(* IEC 61131-3 sources: axftcmlib/src/Sortingline, 10 files *)

(* ---- ISortingline.st ---- *)
NAMESPACE Simatic.Ax.axftcmlib
    INTERFACE ISortingline
        METHOD SlMoveToColorsensor
        END_METHOD
        METHOD SlDetectColor : Bool
        END_METHOD
        METHOD SlMoveToSensor
        END_METHOD
        METHOD SlClearConveyor
        END_METHOD

    END_INTERFACE
END_NAMESPACE

(* ---- Sl1StateIdle.st ---- *)
USING Simatic.Ax.StateFramework;
//SOrtingline is ready for the next Element to be sorted
NAMESPACE Simatic.Ax.axftcmlib

    CLASS INTERNAL SlStateIdle EXTENDS State1Transition
        VAR PUBLIC //Reset
           UsedSortingline : Sortingline;
        END_VAR
        METHOD PUBLIC OVERRIDE  OnEntry
          ;
        END_METHOD
    END_CLASS

END_NAMESPACE

(* ---- Sl2StateMoveToColorSensor.st ---- *)
USING Simatic.Ax.StateFramework;
//If an element is placed infront of the first sensor, the Axis moves to the colorsensor
NAMESPACE Simatic.Ax.axftcmlib

    CLASS INTERNAL SlStateMoveToColorSensor EXTENDS State1Transition
        VAR PUBLIC
          Sortingline : ISortingline;
        END_VAR
        METHOD PUBLIC OVERRIDE  OnEntry
            Sortingline.SlMoveToColorsensor();
        END_METHOD
    END_CLASS

END_NAMESPACE

(* ---- Sl3StateDetectColor-Edit.st ---- *)
USING Simatic.Ax.StateFramework;
//if the axis is done, the sensor detects the color and puts it oput
    //->Color valid PArt will be sorted by pusher -> Path 1
    //->color invalid (=#Unknown) ->Path 2
NAMESPACE Simatic.Ax.axftcmlib

    CLASS INTERNAL SlStateDetectColor EXTENDS State2Transition
    VAR
        UsedSortingline : ISortingline;
    END_VAR
        METHOD PUBLIC OVERRIDE OnEntry
            UsedSortingline.SlDetectColor();
        END_METHOD
    END_CLASS

END_NAMESPACE

(* ---- Sl4_1StateColorDetected.st ---- *)
USING Simatic.Ax.StateFramework;
//Valid element is transported to the next sensor
NAMESPACE Simatic.Ax.axftcmlib

    CLASS INTERNAL SlColorDetected EXTENDS State1Transition
        VAR PUBLIC //Reset
          UsedSortingline : ISortingline;
        END_VAR
        METHOD PUBLIC OVERRIDE  OnEntry
            UsedSortingline.SlMoveToSensor();
        END_METHOD
    END_CLASS

END_NAMESPACE

(* ---- Sl4_2StateColorNotDetected.st ---- *)
USING Simatic.Ax.StateFramework;

//element is thrown out of the Sortingline by the conveyor
NAMESPACE Simatic.Ax.axftcmlib

    CLASS INTERNAL SlColorNotDetected EXTENDS State1Transition
        VAR PUBLIC //Reset
          UsedSortingline : ISortingline;
        END_VAR
        METHOD PUBLIC OVERRIDE  OnEntry
            USedSOrtingline.SlClearConveyor();
        END_METHOD
    END_CLASS

END_NAMESPACE

// SlAxis : AXIS;
// SlVelocity : LREAL;
// Activetime : PULSE := (duration := LT#5.0s);//TODO Duration
// METHOD PUBLIC OVERRIDE  OnEntry
//     VAR
//         dir : INT := 0;
//         Trigger : BOOL;
//     END_VAR
//  Trigger := TRUE;
//  IF ActiveTime.output THEN
//  SlAxis.MoveVelocity(SlVelocity,dir);
//  ELSE
// SlAxis.HALT();
//  END_IF;
// END_METHOD

(* ---- Sl5_1StateChoseCylinder.st ---- *)
USING Simatic.Ax.StateFramework;

NAMESPACE Simatic.Ax.axftcmlib

    CLASS INTERNAL SlChoseCylinder EXTENDS State1Transition
        VAR PUBLIC //Reset
           SlAxis : AXIS;
           SlVelocity : LREAL;
           Sensor : BOOL;
           Color : INT;
           PosWHITE : LINT;
           PosRED : LINT;
           PosBLUE : LINT;

        END_VAR
        METHOD PUBLIC OVERRIDE  OnEntry

            VAR
                value : LINT := 0;
            END_VAR

            IF Sensor = TRUE THEN
                SlAxis.Halt();
                SlAxis.Homing(value);
                IF Color = Colors#WHITE THEN
                    SlAxis.MoveRelative(SlVelocity,PosWHITE);
                ELSIF Color = Colors#RED THEN
                    SlAxis.MoveRelative(SlVelocity, PosRED);
                ELSE
                    SlAxis.MoveRelative(SlVelocity, PosBLUE);
                END_IF;
            END_IF;

        END_METHOD
    END_CLASS

END_NAMESPACE

(* ---- Sl6_1StatePusher.st ---- *)
USING Simatic.Ax.StateFramework;

NAMESPACE Simatic.Ax.axftcmlib

    CLASS INTERNAL SlActivateCylinder EXTENDS State1Transition
        VAR PUBLIC //Reset
            CylinderWhite : PneumaticCylinder;
            CylinderRed : PneumaticCylinder;
            CylinderBlue :  PneumaticCylinder;
           Color : INT;
        END_VAR
        METHOD PUBLIC OVERRIDE  OnEntry
                IF Color = Colors#WHITE THEN
                    CylinderWhite.start();
                ELSIF Color = Colors#RED THEN
                    CylinderRed.start();
                ELSE
                    CylinderBlue.start();
                END_IF;
        END_METHOD
    END_CLASS

END_NAMESPACE

(* ---- Sl71-2SortingDone.st ---- *)
USING Simatic.Ax.StateFramework;

NAMESPACE Simatic.Ax.axftcmlib

    CLASS INTERNAL SlSortingDone EXTENDS State1Transition
        VAR PUBLIC //Reset
           SlAxis : AXIS;
        END_VAR
        METHOD PUBLIC OVERRIDE  OnEntry
               SlAxis.Halt();
        END_METHOD
    END_CLASS

END_NAMESPACE

(* ---- Sortingline.st ---- *)
USING Simatic.Ax.IO;
USING Simatic.Ax.axftcmlib;
USING Simatic.Ax.IO.Output;
USING Simatic.Ax.StateFramework;
USING System.Timer;
NAMESPACE Simatic.Ax.axftcmlib
    CLASS Sortingline EXTENDS ControlModuleAbstract IMPLEMENTS ISortingline

        VAR PUBLIC

            SlAxis : Axis;
            SlTimeProvider : TimeProvider;
            SlAxisVelocity : LREAL;
            SlAxisPositionColorSensor : LINT;
            SlAxisPositionWhite : LINT;
            SlAxisPositionRed : LINT;
            SlAxisPositionBlue : LINT;
            Homingposition : LINT := 0;
            SlColorSensor : ColorSensor;
            SlColorvalue : INT;
            ResultColor : INT;
            ColorArray : ARRAY[0..3] OF ColorRange;
            SlCompressor : PneumaticCompressor;
            SlCoilPushingWhite : IBinOutput;
            SlCoilpushingRed : IBinOutput;
            SlCoilPushingBlue : IBinOutput;
            SlSensorActivation : BOOL;
            SlSensorSorting : BOOL;

            //........
            SlDirection : INT := 0;
            //SlClearTime : LTIME := LT#5s;
           Activetime : PULSE := (duration := LT#5.0s);
        END_VAR

        METHOD PUBLIC SlMoveToColorSensor
           SlAxis.Homing(Homingposition);
           SlAxis.moverelative(SlAxisVelocity, SlAxisPositionColorSensor);
        END_METHOD

        METHOD PUBLIC SlDetectColor : BOOL
            ResultColor :=  SlColorsensor.detectColor(SlColorValue, ColorArray);
            IF ResultColor = Colors#Unknown THEN
                SlDetectColor := FALSE;
            ELSE
                SlDetectColor := TRUE;
            END_IF;
        END_METHOD

        METHOD PUBLIC SlMoveToSensor
            SlAxis.MoveVelocity(SlAxisVelocity, SlDirection);
        END_METHOD

    METHOD PUBLIC SlClearConveyor
        VAR
            Trigger : BOOL;
        END_VAR
             Trigger := TRUE;
             IF ActiveTime.output THEN
                 SlAxis.MoveVelocity(SlAxisVelocity,SlDirection);
             ELSE
                SlAxis.HALT();
             END_IF;
    END_METHOD

        METHOD PROTECTED OVERRIDE RunCyclicCustom
            ;
        END_METHOD

        METHOD PROTECTED OVERRIDE Constructor
            ;
        END_METHOD

    END_CLASS
END_NAMESPACE
